// TIA Portal project "灌装完整程序" (V16)

(* hardware
DEVICE "S7-1200 station_1"  S7-1200 Station
   slot 0: "Rack_0"  S7-1200 Rack  Rack  V1.0
   slot 1: "PLC_1"  CPU 1214C DC/DC/DC  6ES7 214-1AG40-0XB0  V4.4
DEVICE "HMI_1"  TP700 Comfort
   slot 0: "HMI_1"  TP700 Comfort  6AV2 124-0GC01-0AX0  16.0.0.0
   slot 1: "HMI_RT_1"  TP700 Comfort  6AV2 124-0GC01-0AX0  16.0.0.0
   slot 5: "HMI_1.IE_CP_1"  PROFINET Interface  16.0.0.0
      slot 1: "PROFINET Interface_1"  PROFINET Interface
         slot 1: "Port_1"  Port
         slot 2: "Port_2"  Port
   slot 7: "HMI_1.MPI/DP_CP_1"  MPI/DP Interface  16.0.0.0
*)

// ===== PLC "PLC_1"  CPU 1214C DC/DC/DC =====

VAR_GLOBAL   // PLC tag table "默认变量表"
   "System_Byte" AT %MB1 : Byte;
   "FirstScan" AT %M1.0 : Bool;
   "DiagStatusUpdate" AT %M1.1 : Bool;
   "AlwaysTRUE" AT %M1.2 : Bool;
   "AlwaysFALSE" AT %M1.3 : Bool;
   "Clock_Byte" AT %MB0 : Byte;
   "Clock_10Hz" AT %M0.0 : Bool;
   "Clock_5Hz" AT %M0.1 : Bool;
   "Clock_2.5Hz" AT %M0.2 : Bool;
   "Clock_2Hz" AT %M0.3 : Bool;
   "Clock_1.25Hz" AT %M0.4 : Bool;
   "Clock_1Hz" AT %M0.5 : Bool;
   "Clock_0.625Hz" AT %M0.6 : Bool;
   "Clock_0.5Hz" AT %M0.7 : Bool;
END_VAR

VAR_GLOBAL   // PLC tag table "I"
   "启动" AT %I0.0 : Bool;
   "停止" AT %I0.1 : Bool;
   "到达称重吹气位置" AT %I0.2 : Bool;
   "到达灌装位置" AT %I0.3 : Bool;
   "到达拧盖位置" AT %I0.4 : Bool;
   "到达包装热缩位置" AT %I0.5 : Bool;
   "到达清洗位置" AT %I0.6 : Bool;
   "到达消毒位置" AT %I0.7 : Bool;
   "到达标签投放位置" AT %I1.0 : Bool;
   "称重检测" AT %IW30 : Int;
   "液位检测" AT %IW32 : Int;
   "吹气气缸上限位" AT %I1.1 : Bool;
   "吹气气缸下限位" AT %I1.2 : Bool;
   "灌装气缸上限位" AT %I1.3 : Bool;
   "灌装气缸下限位" AT %I1.4 : Bool;
   "拧盖气缸上限位" AT %I1.5 : Bool;
   "拧盖气缸下限位" AT %I2.0 : Bool;
   "复位" AT %I2.1 : Bool;
END_VAR

VAR_GLOBAL   // PLC tag table "O"
   "运行指示灯" AT %Q0.0 : Bool;
   "吹气阀门" AT %Q0.1 : Bool;
   "灌装阀门" AT %Q0.2 : Bool;
   "拧盖气缸" AT %Q0.3 : Bool;
   "拧盖电机" AT %Q0.4 : Bool;
   "标签投放" AT %Q0.5 : Bool;
   "包装热缩" AT %Q0.6 : Bool;
   "清洗机" AT %Q0.7 : Bool;
   "消毒机" AT %Q1.0 : Bool;
   "传送带" AT %Q1.1 : Bool;
   "吹气气缸" AT %Q2.0 : Bool;
   "灌装气缸" AT %Q2.1 : Bool;
   "瓶子异常示灯" AT %Q2.2 : Bool;
   "有杂物指示灯" AT %Q2.3 : Bool;
END_VAR

DATA_BLOCK "DB"   // DB1
{ S7_Optimized_Access := 'TRUE' }
VERSION : 0.1
   VAR
      "P/N" : Array[0..100] of Bool;
      仿真数据 : Struct
         仿真开关 : Bool;
         传送带 : Int;
         罐子 : Struct
            X : Int;
            Y : Int;
         END_STRUCT;
         吹气 : Struct
            气缸 : Int;
         END_STRUCT;
         灌装 : Struct
            气缸 : Int;
            液位 : Int;
         END_STRUCT;
         拧盖 : Struct
            盖子显示 : Bool;
            气缸 : Int;
            拧盖进度 : Int;
         END_STRUCT;
         标签投放 : Struct
            大标显示 : Bool;
            小标显示 : Bool;
            标签X : Int;
            标签Y : Int;
            标签Y辅助 : Int;
         END_STRUCT;
         热缩 : Struct
            热缩进度 : Int;
         END_STRUCT;
         清洗 : Struct
            清洗进度 : Int;
         END_STRUCT;
         消毒 : Struct
            消毒进度 : Int;
         END_STRUCT;
      END_STRUCT;
      HMI按键 : Struct
         启动 : Bool;
         停止 : Bool;
         复位 : Bool;
         仿真瓶子质量过低 : Bool;
         仿真瓶子质量超重 : Bool;
      END_STRUCT;
      设定数据 : Struct
         称重质量上限 : Real := 160.0;
         称重质量下限 : Real := 140.0;
         灌装液位 : Int := 85;
      END_STRUCT;
      检测数据 : Struct
         转换值 : Array[0..1] of Real;
         中间值 : Array[0..1] of Real;
         液位实际值 : Real;
         称重实际值 : Real;
         液位仿真值 : Real;
         称重仿真值 : Real;
      END_STRUCT;
      状态 : Struct
         完成吹气 : Bool;
         吹气气缸缩回 : Bool;
         完成灌装 : Bool;
         灌装气缸缩回 : Bool;
         完成拧盖 : Bool;
         拧盖气缸缩回 : Bool;
         标签投放完毕 : Bool;
         热缩完毕 : Bool;
         清洗完毕 : Bool;
         消毒完毕 : Bool;
         流程 : Int;
      END_STRUCT;
   END_VAR
BEGIN
END_DATA_BLOCK

// folder: System blocks/Program resources

DATA_BLOCK "IEC_Timer_0_DB"   // DB2
{ S7_Optimized_Access := 'TRUE' }
AUTHOR : Simatic
FAMILY : IEC
NAME : IEC_TMR
VERSION : 1.0
// stored: InstanceOfName IEC_TIMER
"IEC_TIMER"
BEGIN
END_DATA_BLOCK

DATA_BLOCK "IEC_Timer_0_DB_1"   // DB3
{ S7_Optimized_Access := 'TRUE' }
AUTHOR : Simatic
FAMILY : IEC
NAME : IEC_TMR
VERSION : 1.0
// stored: InstanceOfName IEC_TIMER
"IEC_TIMER"
BEGIN
END_DATA_BLOCK

DATA_BLOCK "IEC_Timer_0_DB_2"   // DB4
{ S7_Optimized_Access := 'TRUE' }
AUTHOR : Simatic
FAMILY : IEC
NAME : IEC_TMR
VERSION : 1.0
// stored: InstanceOfName IEC_TIMER
"IEC_TIMER"
BEGIN
END_DATA_BLOCK

DATA_BLOCK "IEC_Timer_0_DB_3"   // DB5
{ S7_Optimized_Access := 'TRUE' }
AUTHOR : Simatic
FAMILY : IEC
NAME : IEC_TMR
VERSION : 1.0
// stored: InstanceOfName IEC_TIMER
"IEC_TIMER"
BEGIN
END_DATA_BLOCK

DATA_BLOCK "吹气延时"   // DB6
{ S7_Optimized_Access := 'TRUE' }
AUTHOR : Simatic
FAMILY : IEC
NAME : IEC_TMR
VERSION : 1.0
// stored: InstanceOfName IEC_TIMER
"IEC_TIMER"
BEGIN
END_DATA_BLOCK

// folder: (top level)

FUNCTION "04流程" : Void   // FC1, LAD
{ S7_Optimized_Access := 'TRUE' }
VERSION : 0.1
BEGIN

REGION Network 1
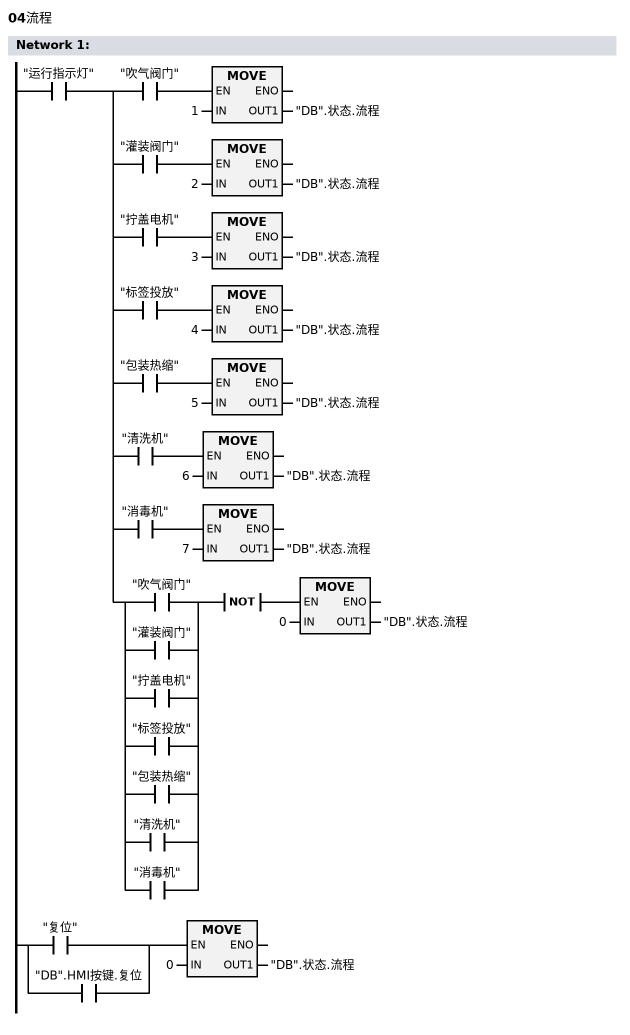
   RUNG wire#powerrail
      Contact( "运行指示灯" )
      wire#w1
      Contact( "吹气阀门" )
      Move(in := 1, out1 => "DB".状态.流程)
   END_RUNG
   RUNG wire#w1
      Contact( "灌装阀门" )
      Move(in := 2, out1 => "DB".状态.流程)
   END_RUNG
   RUNG wire#w1
      Contact( "拧盖电机" )
      Move(in := 3, out1 => "DB".状态.流程)
   END_RUNG
   RUNG wire#w1
      Contact( "标签投放" )
      Move(in := 4, out1 => "DB".状态.流程)
   END_RUNG
   RUNG wire#w1
      Contact( "包装热缩" )
      Move(in := 5, out1 => "DB".状态.流程)
   END_RUNG
   RUNG wire#w1
      Contact( "清洗机" )
      Move(in := 6, out1 => "DB".状态.流程)
   END_RUNG
   RUNG wire#w1
      Contact( "消毒机" )
      Move(in := 7, out1 => "DB".状态.流程)
   END_RUNG
   RUNG wire#w1
      Contact( "吹气阀门" )
      wire#w2
      Not()
      Move(in := 0, out1 => "DB".状态.流程)
   END_RUNG
   RUNG wire#w1
      Contact( "灌装阀门" )
   END_RUNG wire#w2
   RUNG wire#w1
      Contact( "拧盖电机" )
   END_RUNG wire#w2
   RUNG wire#w1
      Contact( "标签投放" )
   END_RUNG wire#w2
   RUNG wire#w1
      Contact( "包装热缩" )
   END_RUNG wire#w2
   RUNG wire#w1
      Contact( "清洗机" )
   END_RUNG wire#w2
   RUNG wire#w1
      Contact( "消毒机" )
   END_RUNG wire#w2
   RUNG wire#powerrail
      Contact( "复位" )
      wire#w3
      Move(in := 0, out1 => "DB".状态.流程)
   END_RUNG
   RUNG wire#powerrail
      Contact( "DB".HMI按键.复位 )
   END_RUNG wire#w3
   // the same network as SCL:
   IF "运行指示灯" AND "吹气阀门" THEN "DB".状态.流程 := 1; END_IF;
   IF "运行指示灯" AND "灌装阀门" THEN "DB".状态.流程 := 2; END_IF;
   IF "运行指示灯" AND "拧盖电机" THEN "DB".状态.流程 := 3; END_IF;
   IF "运行指示灯" AND "标签投放" THEN "DB".状态.流程 := 4; END_IF;
   IF "运行指示灯" AND "包装热缩" THEN "DB".状态.流程 := 5; END_IF;
   IF "运行指示灯" AND "清洗机" THEN "DB".状态.流程 := 6; END_IF;
   IF "运行指示灯" AND "消毒机" THEN "DB".状态.流程 := 7; END_IF;
   IF NOT ("运行指示灯" AND ("吹气阀门" OR "灌装阀门" OR "拧盖电机" OR "标签投放" OR "包装热缩" OR "清洗机" OR "消毒机")) THEN
       "DB".状态.流程 := 0;
   END_IF;
   IF "复位" OR "DB".HMI按键.复位 THEN "DB".状态.流程 := 0; END_IF;
END_REGION
END_FUNCTION

FUNCTION "01系统启停" : Void   // FC2, LAD
{ S7_Optimized_Access := 'TRUE' }
VERSION : 0.1
BEGIN

REGION Network 1
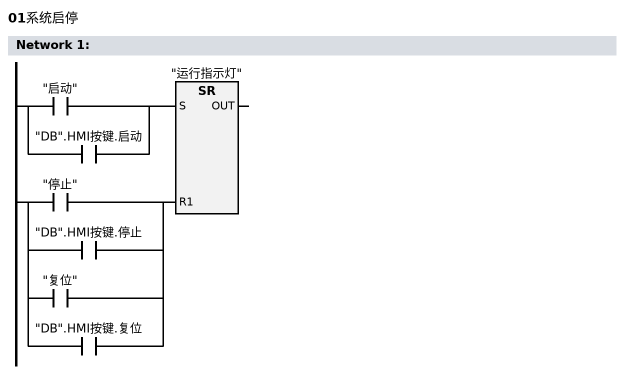
   RUNG wire#powerrail
      Contact( "启动" )
      wire#w1
      S_SR(operand := "运行指示灯", r1 := wire#w2)
   END_RUNG
   RUNG wire#powerrail
      Contact( "DB".HMI按键.启动 )
   END_RUNG wire#w1
   RUNG wire#powerrail
      Contact( "停止" )
   END_RUNG wire#w2
   RUNG wire#powerrail
      Contact( "DB".HMI按键.停止 )
   END_RUNG wire#w2
   RUNG wire#powerrail
      Contact( "复位" )
   END_RUNG wire#w2
   RUNG wire#powerrail
      Contact( "DB".HMI按键.复位 )
   END_RUNG wire#w2
   // the same network as SCL:
   IF "启动" OR "DB".HMI按键.启动 THEN
       "运行指示灯" := TRUE;   // SR flip-flop
   END_IF;
   IF "停止" OR "DB".HMI按键.停止 OR "复位" OR "DB".HMI按键.复位 THEN "运行指示灯" := FALSE; END_IF;
END_REGION
END_FUNCTION

FUNCTION "03自动控制部分" : Void   // FC3, LAD
{ S7_Optimized_Access := 'TRUE' }
VERSION : 0.1
   VAR_TEMP   // added for the SCL form of the ladder/FBD networks
      _w1 : Bool;
      _w2 : Bool;
      _w3 : Bool;
   END_VAR
BEGIN

REGION Network 1
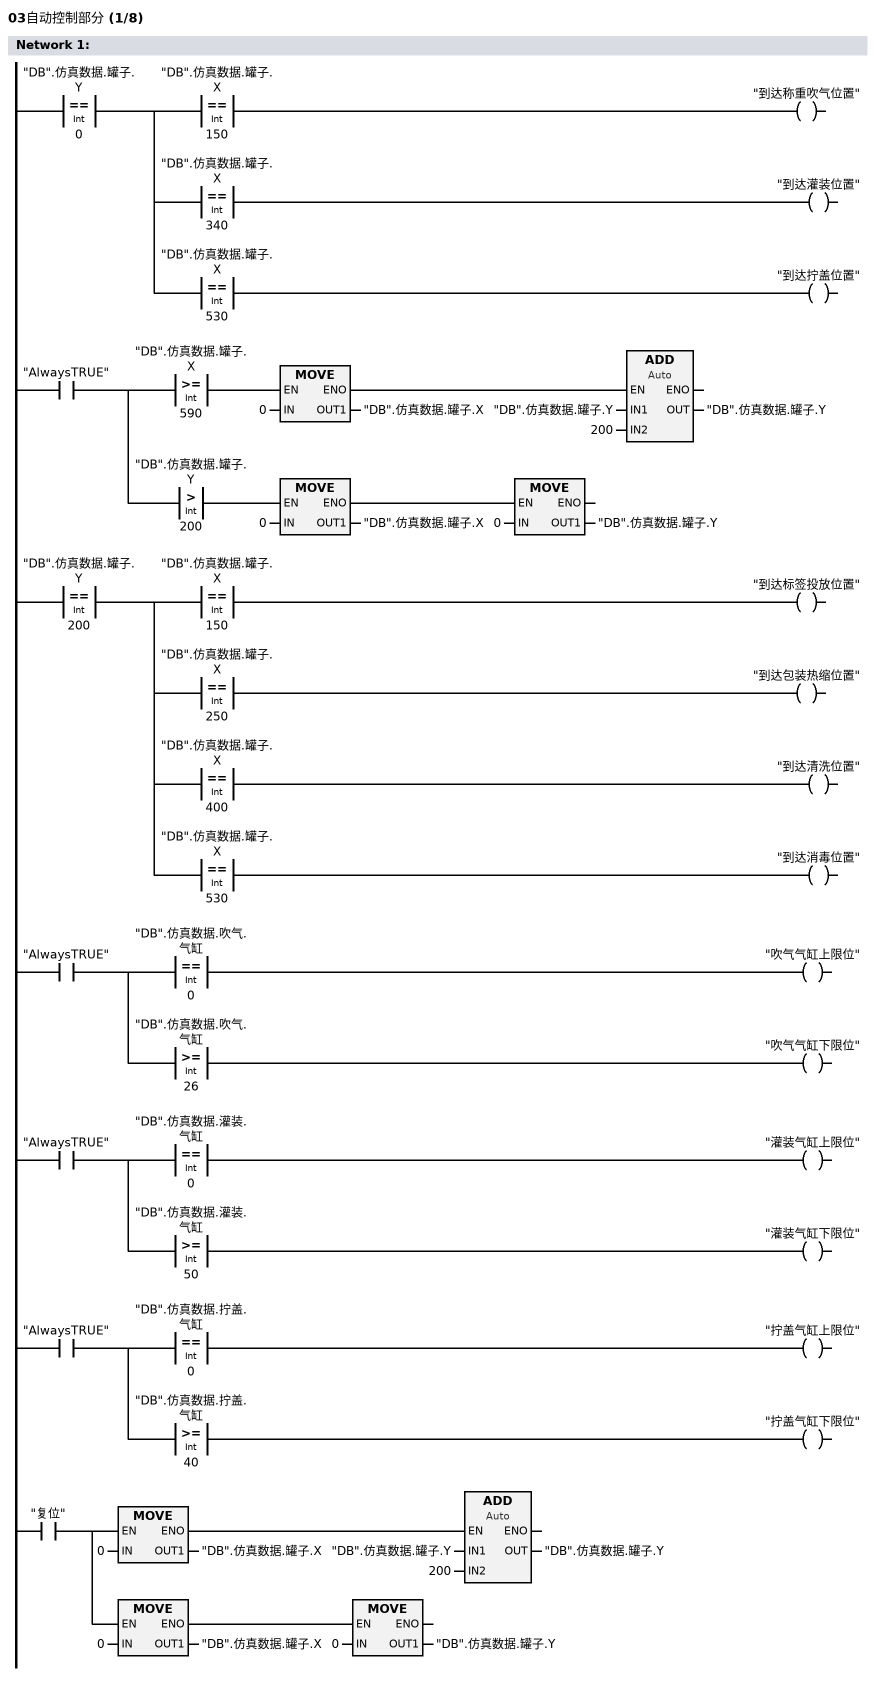
   RUNG wire#powerrail
      { S7_Templates := "SrcType := Int" } EQ_Contact(in1 := "DB".仿真数据.罐子.Y, in2 := 0)
      wire#w1
      { S7_Templates := "SrcType := Int" } EQ_Contact(in1 := "DB".仿真数据.罐子.X, in2 := 150)
      Coil( "到达称重吹气位置" )
   END_RUNG
   RUNG wire#w1
      { S7_Templates := "SrcType := Int" } EQ_Contact(in1 := "DB".仿真数据.罐子.X, in2 := 340)
      Coil( "到达灌装位置" )
   END_RUNG
   RUNG wire#w1
      { S7_Templates := "SrcType := Int" } EQ_Contact(in1 := "DB".仿真数据.罐子.X, in2 := 530)
      Coil( "到达拧盖位置" )
   END_RUNG
   RUNG wire#powerrail
      Contact( "AlwaysTRUE" )
      wire#w2
      { S7_Templates := "SrcType := Int" } GE_Contact(in1 := "DB".仿真数据.罐子.X, in2 := 590)
      Move(in := 0, out1 => "DB".仿真数据.罐子.X)
      Add(in1 := "DB".仿真数据.罐子.Y, in2 := 200, out => "DB".仿真数据.罐子.Y)
   END_RUNG
   RUNG wire#w2
      { S7_Templates := "SrcType := Int" } GT_Contact(in1 := "DB".仿真数据.罐子.Y, in2 := 200)
      Move(in := 0, out1 => "DB".仿真数据.罐子.X)
      Move(in := 0, out1 => "DB".仿真数据.罐子.Y)
   END_RUNG
   RUNG wire#powerrail
      { S7_Templates := "SrcType := Int" } EQ_Contact(in1 := "DB".仿真数据.罐子.Y, in2 := 200)
      wire#w3
      { S7_Templates := "SrcType := Int" } EQ_Contact(in1 := "DB".仿真数据.罐子.X, in2 := 150)
      Coil( "到达标签投放位置" )
   END_RUNG
   RUNG wire#w3
      { S7_Templates := "SrcType := Int" } EQ_Contact(in1 := "DB".仿真数据.罐子.X, in2 := 250)
      Coil( "到达包装热缩位置" )
   END_RUNG
   RUNG wire#w3
      { S7_Templates := "SrcType := Int" } EQ_Contact(in1 := "DB".仿真数据.罐子.X, in2 := 400)
      Coil( "到达清洗位置" )
   END_RUNG
   RUNG wire#w3
      { S7_Templates := "SrcType := Int" } EQ_Contact(in1 := "DB".仿真数据.罐子.X, in2 := 530)
      Coil( "到达消毒位置" )
   END_RUNG
   RUNG wire#powerrail
      Contact( "AlwaysTRUE" )
      wire#w4
      { S7_Templates := "SrcType := Int" } EQ_Contact(in1 := "DB".仿真数据.吹气.气缸, in2 := 0)
      Coil( "吹气气缸上限位" )
   END_RUNG
   RUNG wire#w4
      { S7_Templates := "SrcType := Int" } GE_Contact(in1 := "DB".仿真数据.吹气.气缸, in2 := 26)
      Coil( "吹气气缸下限位" )
   END_RUNG
   RUNG wire#powerrail
      Contact( "AlwaysTRUE" )
      wire#w5
      { S7_Templates := "SrcType := Int" } EQ_Contact(in1 := "DB".仿真数据.灌装.气缸, in2 := 0)
      Coil( "灌装气缸上限位" )
   END_RUNG
   RUNG wire#w5
      { S7_Templates := "SrcType := Int" } GE_Contact(in1 := "DB".仿真数据.灌装.气缸, in2 := 50)
      Coil( "灌装气缸下限位" )
   END_RUNG
   RUNG wire#powerrail
      Contact( "AlwaysTRUE" )
      wire#w6
      { S7_Templates := "SrcType := Int" } EQ_Contact(in1 := "DB".仿真数据.拧盖.气缸, in2 := 0)
      Coil( "拧盖气缸上限位" )
   END_RUNG
   RUNG wire#w6
      { S7_Templates := "SrcType := Int" } GE_Contact(in1 := "DB".仿真数据.拧盖.气缸, in2 := 40)
      Coil( "拧盖气缸下限位" )
   END_RUNG
   RUNG wire#powerrail
      Contact( "复位" )
      wire#w7
      Move(in := 0, out1 => "DB".仿真数据.罐子.X)
      Add(in1 := "DB".仿真数据.罐子.Y, in2 := 200, out => "DB".仿真数据.罐子.Y)
   END_RUNG
   RUNG wire#w7
      Move(in := 0, out1 => "DB".仿真数据.罐子.X)
      Move(in := 0, out1 => "DB".仿真数据.罐子.Y)
   END_RUNG
   // the same network as SCL:
   #_w1 := "DB".仿真数据.罐子.Y = 0;
   "到达称重吹气位置" := #_w1 AND ("DB".仿真数据.罐子.X = 150);
   "到达灌装位置" := #_w1 AND ("DB".仿真数据.罐子.X = 340);
   "到达拧盖位置" := #_w1 AND ("DB".仿真数据.罐子.X = 530);
   #_w2 := "AlwaysTRUE" AND ("DB".仿真数据.罐子.X >= 590);
   IF #_w2 THEN
       "DB".仿真数据.罐子.X := 0;
       "DB".仿真数据.罐子.Y := "DB".仿真数据.罐子.Y + 200;
   END_IF;
   IF "AlwaysTRUE" AND ("DB".仿真数据.罐子.Y > 200) THEN
       "DB".仿真数据.罐子.X := 0;
       "DB".仿真数据.罐子.Y := 0;
   END_IF;
   #_w3 := "DB".仿真数据.罐子.Y = 200;
   "到达标签投放位置" := #_w3 AND ("DB".仿真数据.罐子.X = 150);
   "到达包装热缩位置" := #_w3 AND ("DB".仿真数据.罐子.X = 250);
   "到达清洗位置" := #_w3 AND ("DB".仿真数据.罐子.X = 400);
   "到达消毒位置" := #_w3 AND ("DB".仿真数据.罐子.X = 530);
   "吹气气缸上限位" := "AlwaysTRUE" AND ("DB".仿真数据.吹气.气缸 = 0);
   "吹气气缸下限位" := "AlwaysTRUE" AND ("DB".仿真数据.吹气.气缸 >= 26);
   "灌装气缸上限位" := "AlwaysTRUE" AND ("DB".仿真数据.灌装.气缸 = 0);
   "灌装气缸下限位" := "AlwaysTRUE" AND ("DB".仿真数据.灌装.气缸 >= 50);
   "拧盖气缸上限位" := "AlwaysTRUE" AND ("DB".仿真数据.拧盖.气缸 = 0);
   "拧盖气缸下限位" := "AlwaysTRUE" AND ("DB".仿真数据.拧盖.气缸 >= 40);
   IF "复位" THEN
       "DB".仿真数据.罐子.X := 0;
       "DB".仿真数据.罐子.Y := "DB".仿真数据.罐子.Y + 200;
       "DB".仿真数据.罐子.X := 0;
       "DB".仿真数据.罐子.Y := 0;
   END_IF;
END_REGION

REGION Network 2: 传送带控制
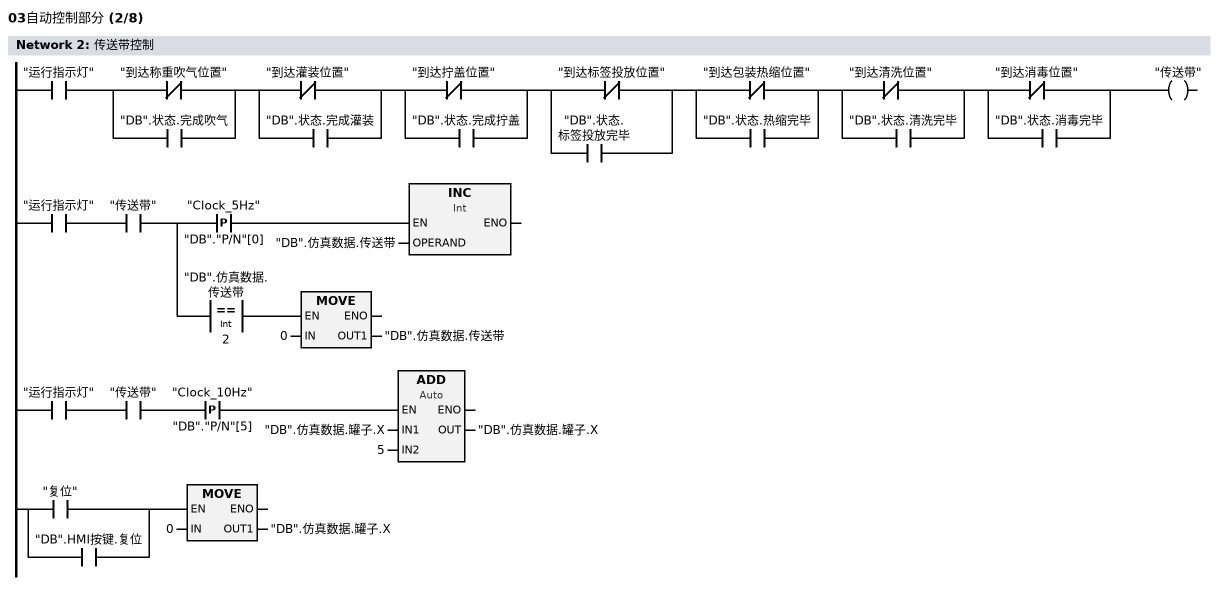
   RUNG wire#powerrail
      Contact( "运行指示灯" )
      wire#w1
      I_Contact( "到达称重吹气位置" )
      wire#w2
      I_Contact( "到达灌装位置" )
      wire#w3
      I_Contact( "到达拧盖位置" )
      wire#w4
      I_Contact( "到达标签投放位置" )
      wire#w5
      I_Contact( "到达包装热缩位置" )
      wire#w6
      I_Contact( "到达清洗位置" )
      wire#w7
      I_Contact( "到达消毒位置" )
      wire#w8
      Coil( "传送带" )
   END_RUNG
   RUNG wire#w1
      Contact( "DB".状态.完成吹气 )
   END_RUNG wire#w2
   RUNG wire#w2
      Contact( "DB".状态.完成灌装 )
   END_RUNG wire#w3
   RUNG wire#w3
      Contact( "DB".状态.完成拧盖 )
   END_RUNG wire#w4
   RUNG wire#w4
      Contact( "DB".状态.标签投放完毕 )
   END_RUNG wire#w5
   RUNG wire#w5
      Contact( "DB".状态.热缩完毕 )
   END_RUNG wire#w6
   RUNG wire#w6
      Contact( "DB".状态.清洗完毕 )
   END_RUNG wire#w7
   RUNG wire#w7
      Contact( "DB".状态.消毒完毕 )
   END_RUNG wire#w8
   RUNG wire#powerrail
      Contact( "运行指示灯" )
      Contact( "传送带" )
      wire#w9
      P_Contact(operand := "Clock_5Hz", bit := "DB"."P/N"[0])
      { S7_Templates := "DestType := Int" } Inc( "DB".仿真数据.传送带 )
   END_RUNG
   RUNG wire#w9
      { S7_Templates := "SrcType := Int" } EQ_Contact(in1 := "DB".仿真数据.传送带, in2 := 2)
      Move(in := 0, out1 => "DB".仿真数据.传送带)
   END_RUNG
   RUNG wire#powerrail
      Contact( "运行指示灯" )
      Contact( "传送带" )
      P_Contact(operand := "Clock_10Hz", bit := "DB"."P/N"[5])
      Add(in1 := "DB".仿真数据.罐子.X, in2 := 5, out => "DB".仿真数据.罐子.X)
   END_RUNG
   RUNG wire#powerrail
      Contact( "复位" )
      wire#w10
      Move(in := 0, out1 => "DB".仿真数据.罐子.X)
   END_RUNG
   RUNG wire#powerrail
      Contact( "DB".HMI按键.复位 )
   END_RUNG wire#w10
   // the same network as SCL:
   "传送带" := "运行指示灯" AND (NOT "到达称重吹气位置" OR "DB".状态.完成吹气) AND (NOT "到达灌装位置" OR "DB".状态.完成灌装) AND (NOT "到达拧盖位置" OR "DB".状态.完成拧盖) AND (NOT "到达标签投放位置" OR "DB".状态.标签投放完毕) AND (NOT "到达包装热缩位置" OR "DB".状态.热缩完毕) AND (NOT "到达清洗位置" OR "DB".状态.清洗完毕) AND (NOT "到达消毒位置" OR "DB".状态.消毒完毕);
   #_w1 := "运行指示灯" AND "传送带";
   #_w2 := #_w1 AND "Clock_5Hz" AND NOT "DB"."P/N"[0];   // rising edge of "Clock_5Hz"
   "DB"."P/N"[0] := "Clock_5Hz";
   IF #_w2 THEN "DB".仿真数据.传送带 := "DB".仿真数据.传送带 + 1; END_IF;
   IF #_w1 AND ("DB".仿真数据.传送带 = 2) THEN "DB".仿真数据.传送带 := 0; END_IF;
   #_w3 := "运行指示灯" AND "传送带" AND "Clock_10Hz" AND NOT "DB"."P/N"[5];   // rising edge of "Clock_10Hz"
   "DB"."P/N"[5] := "Clock_10Hz";
   IF #_w3 THEN "DB".仿真数据.罐子.X := "DB".仿真数据.罐子.X + 5; END_IF;
   IF "复位" OR "DB".HMI按键.复位 THEN "DB".仿真数据.罐子.X := 0; END_IF;
END_REGION

REGION Network 3: 称重吹气
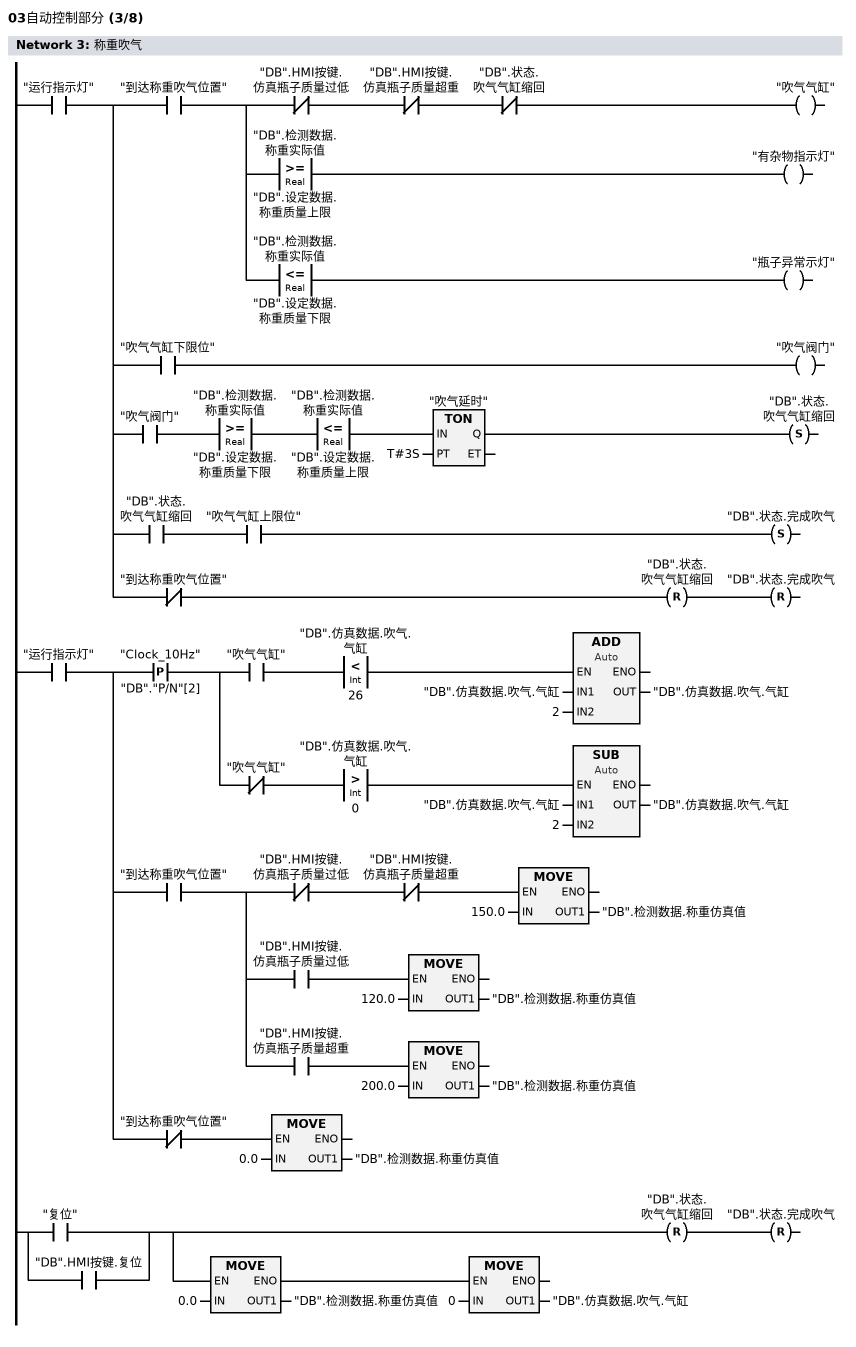
   #_w1 := "运行指示灯" AND "到达称重吹气位置";
   "吹气气缸" := #_w1 AND NOT "DB".HMI按键.仿真瓶子质量过低 AND NOT "DB".HMI按键.仿真瓶子质量超重 AND NOT "DB".状态.吹气气缸缩回;
   "有杂物指示灯" := #_w1 AND ("DB".检测数据.称重实际值 >= "DB".设定数据.称重质量上限);
   "瓶子异常示灯" := #_w1 AND ("DB".检测数据.称重实际值 <= "DB".设定数据.称重质量下限);
   "吹气阀门" := "运行指示灯" AND "吹气气缸下限位";
   "吹气延时".TON(IN := "运行指示灯" AND "吹气阀门" AND ("DB".检测数据.称重实际值 >= "DB".设定数据.称重质量下限) AND ("DB".检测数据.称重实际值 <= "DB".设定数据.称重质量上限),
              PT := T#3S);
   IF "吹气延时".Q THEN "DB".状态.吹气气缸缩回 := TRUE; END_IF;
   IF "运行指示灯" AND "DB".状态.吹气气缸缩回 AND "吹气气缸上限位" THEN "DB".状态.完成吹气 := TRUE; END_IF;
   IF "运行指示灯" AND NOT "到达称重吹气位置" THEN
       "DB".状态.吹气气缸缩回 := FALSE;
       "DB".状态.完成吹气 := FALSE;
   END_IF;
   #_w2 := "运行指示灯" AND "Clock_10Hz" AND NOT "DB"."P/N"[2];   // rising edge of "Clock_10Hz"
   "DB"."P/N"[2] := "Clock_10Hz";
   IF #_w2 AND "吹气气缸" AND ("DB".仿真数据.吹气.气缸 < 26) THEN "DB".仿真数据.吹气.气缸 := "DB".仿真数据.吹气.气缸 + 2; END_IF;
   IF #_w2 AND NOT "吹气气缸" AND ("DB".仿真数据.吹气.气缸 > 0) THEN "DB".仿真数据.吹气.气缸 := "DB".仿真数据.吹气.气缸 - 2; END_IF;
   #_w3 := "运行指示灯" AND "到达称重吹气位置";
   IF #_w3 AND NOT "DB".HMI按键.仿真瓶子质量过低 AND NOT "DB".HMI按键.仿真瓶子质量超重 THEN "DB".检测数据.称重仿真值 := 150.0; END_IF;
   IF #_w3 AND "DB".HMI按键.仿真瓶子质量过低 THEN "DB".检测数据.称重仿真值 := 120.0; END_IF;
   IF #_w3 AND "DB".HMI按键.仿真瓶子质量超重 THEN "DB".检测数据.称重仿真值 := 200.0; END_IF;
   IF "运行指示灯" AND NOT "到达称重吹气位置" THEN "DB".检测数据.称重仿真值 := 0.0; END_IF;
   IF "复位" OR "DB".HMI按键.复位 THEN
       "DB".状态.吹气气缸缩回 := FALSE;
       "DB".状态.完成吹气 := FALSE;
       "DB".检测数据.称重仿真值 := 0.0;
       "DB".仿真数据.吹气.气缸 := 0;
   END_IF;
END_REGION

REGION Network 4: 灌装
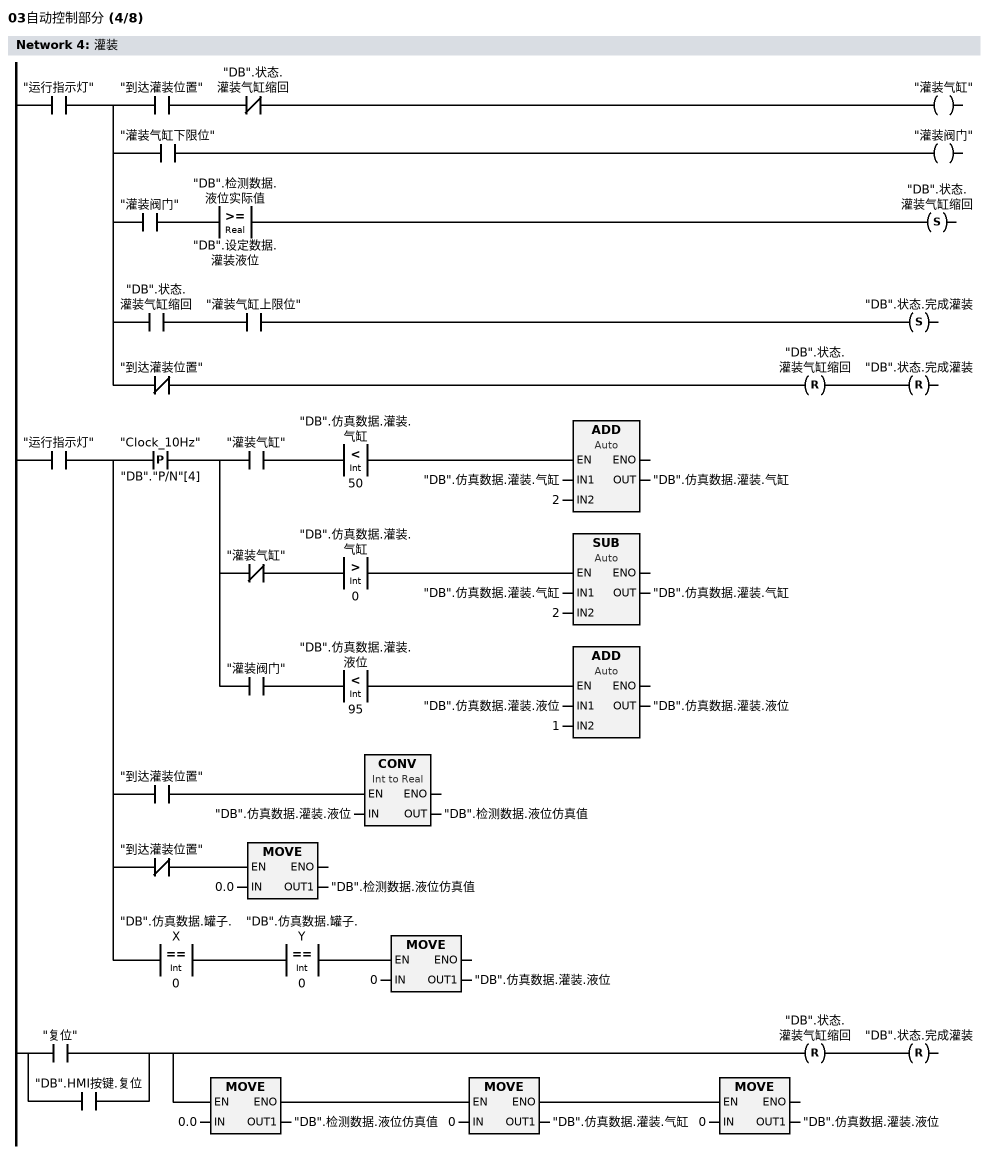
   RUNG wire#powerrail
      Contact( "运行指示灯" )
      wire#w1
      Contact( "到达灌装位置" )
      I_Contact( "DB".状态.灌装气缸缩回 )
      Coil( "灌装气缸" )
   END_RUNG
   RUNG wire#w1
      Contact( "灌装气缸下限位" )
      Coil( "灌装阀门" )
   END_RUNG
   RUNG wire#w1
      Contact( "灌装阀门" )
      { S7_Templates := "SrcType := Real" } GE_Contact(in1 := "DB".检测数据.液位实际值, in2 := "DB".设定数据.灌装液位)
      S_Coil( "DB".状态.灌装气缸缩回 )
   END_RUNG
   RUNG wire#w1
      Contact( "DB".状态.灌装气缸缩回 )
      Contact( "灌装气缸上限位" )
      S_Coil( "DB".状态.完成灌装 )
   END_RUNG
   RUNG wire#w1
      I_Contact( "到达灌装位置" )
      R_Coil( "DB".状态.灌装气缸缩回 )
      R_Coil( "DB".状态.完成灌装 )
   END_RUNG
   RUNG wire#powerrail
      Contact( "运行指示灯" )
      wire#w2
      P_Contact(operand := "Clock_10Hz", bit := "DB"."P/N"[4])
      wire#w3
      Contact( "灌装气缸" )
      { S7_Templates := "SrcType := Int" } LT_Contact(in1 := "DB".仿真数据.灌装.气缸, in2 := 50)
      Add(in1 := "DB".仿真数据.灌装.气缸, in2 := 2, out => "DB".仿真数据.灌装.气缸)
   END_RUNG
   RUNG wire#w3
      I_Contact( "灌装气缸" )
      { S7_Templates := "SrcType := Int" } GT_Contact(in1 := "DB".仿真数据.灌装.气缸, in2 := 0)
      Sub(in1 := "DB".仿真数据.灌装.气缸, in2 := 2, out => "DB".仿真数据.灌装.气缸)
   END_RUNG
   RUNG wire#w3
      Contact( "灌装阀门" )
      { S7_Templates := "SrcType := Int" } LT_Contact(in1 := "DB".仿真数据.灌装.液位, in2 := 95)
      Add(in1 := "DB".仿真数据.灌装.液位, in2 := 1, out => "DB".仿真数据.灌装.液位)
   END_RUNG
   RUNG wire#w2
      Contact( "到达灌装位置" )
      { S7_Templates := "[SrcType := Int, DestType := Real]" } Convert(in := "DB".仿真数据.灌装.液位, out => "DB".检测数据.液位仿真值)
   END_RUNG
   RUNG wire#w2
      I_Contact( "到达灌装位置" )
      Move(in := 0.0, out1 => "DB".检测数据.液位仿真值)
   END_RUNG
   RUNG wire#w2
      { S7_Templates := "SrcType := Int" } EQ_Contact(in1 := "DB".仿真数据.罐子.X, in2 := 0)
      { S7_Templates := "SrcType := Int" } EQ_Contact(in1 := "DB".仿真数据.罐子.Y, in2 := 0)
      Move(in := 0, out1 => "DB".仿真数据.灌装.液位)
   END_RUNG
   RUNG wire#powerrail
      Contact( "复位" )
      wire#w4
      R_Coil( "DB".状态.灌装气缸缩回 )
      R_Coil( "DB".状态.完成灌装 )
   END_RUNG
   RUNG wire#powerrail
      Contact( "DB".HMI按键.复位 )
   END_RUNG wire#w4
   RUNG wire#w4
      Move(in := 0.0, out1 => "DB".检测数据.液位仿真值)
      Move(in := 0, out1 => "DB".仿真数据.灌装.气缸)
      Move(in := 0, out1 => "DB".仿真数据.灌装.液位)
   END_RUNG
   // the same network as SCL:
   "灌装气缸" := "运行指示灯" AND "到达灌装位置" AND NOT "DB".状态.灌装气缸缩回;
   "灌装阀门" := "运行指示灯" AND "灌装气缸下限位";
   IF "运行指示灯" AND "灌装阀门" AND ("DB".检测数据.液位实际值 >= "DB".设定数据.灌装液位) THEN "DB".状态.灌装气缸缩回 := TRUE; END_IF;
   IF "运行指示灯" AND "DB".状态.灌装气缸缩回 AND "灌装气缸上限位" THEN "DB".状态.完成灌装 := TRUE; END_IF;
   IF "运行指示灯" AND NOT "到达灌装位置" THEN
       "DB".状态.灌装气缸缩回 := FALSE;
       "DB".状态.完成灌装 := FALSE;
   END_IF;
   #_w1 := "运行指示灯" AND "Clock_10Hz" AND NOT "DB"."P/N"[4];   // rising edge of "Clock_10Hz"
   "DB"."P/N"[4] := "Clock_10Hz";
   IF #_w1 AND "灌装气缸" AND ("DB".仿真数据.灌装.气缸 < 50) THEN "DB".仿真数据.灌装.气缸 := "DB".仿真数据.灌装.气缸 + 2; END_IF;
   IF #_w1 AND NOT "灌装气缸" AND ("DB".仿真数据.灌装.气缸 > 0) THEN "DB".仿真数据.灌装.气缸 := "DB".仿真数据.灌装.气缸 - 2; END_IF;
   IF #_w1 AND "灌装阀门" AND ("DB".仿真数据.灌装.液位 < 95) THEN "DB".仿真数据.灌装.液位 := "DB".仿真数据.灌装.液位 + 1; END_IF;
   IF "运行指示灯" AND "到达灌装位置" THEN "DB".检测数据.液位仿真值 := INT_TO_REAL("DB".仿真数据.灌装.液位); END_IF;
   IF "运行指示灯" AND NOT "到达灌装位置" THEN "DB".检测数据.液位仿真值 := 0.0; END_IF;
   IF "运行指示灯" AND ("DB".仿真数据.罐子.X = 0) AND ("DB".仿真数据.罐子.Y = 0) THEN "DB".仿真数据.灌装.液位 := 0; END_IF;
   IF "复位" OR "DB".HMI按键.复位 THEN
       "DB".状态.灌装气缸缩回 := FALSE;
       "DB".状态.完成灌装 := FALSE;
       "DB".检测数据.液位仿真值 := 0.0;
       "DB".仿真数据.灌装.气缸 := 0;
       "DB".仿真数据.灌装.液位 := 0;
   END_IF;
END_REGION

REGION Network 5: 拧盖
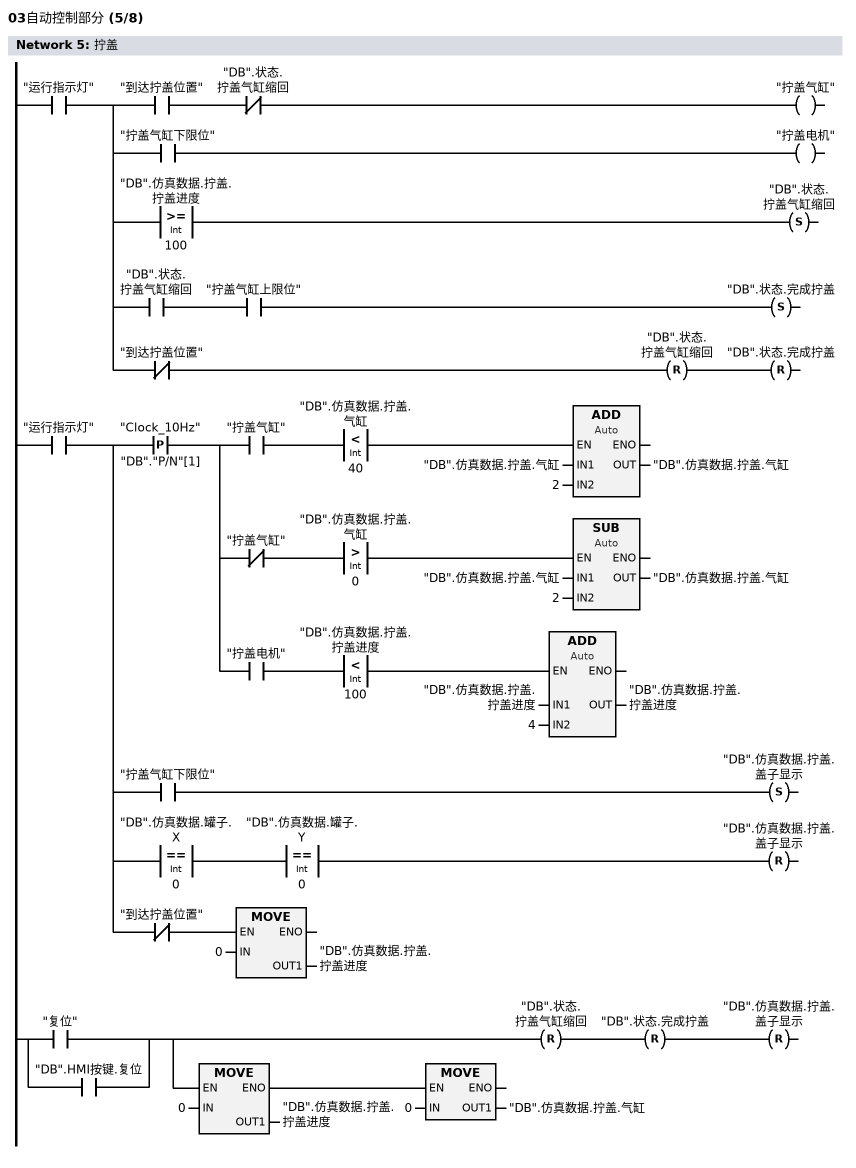
   RUNG wire#powerrail
      Contact( "运行指示灯" )
      wire#w1
      Contact( "到达拧盖位置" )
      I_Contact( "DB".状态.拧盖气缸缩回 )
      Coil( "拧盖气缸" )
   END_RUNG
   RUNG wire#w1
      Contact( "拧盖气缸下限位" )
      Coil( "拧盖电机" )
   END_RUNG
   RUNG wire#w1
      { S7_Templates := "SrcType := Int" } GE_Contact(in1 := "DB".仿真数据.拧盖.拧盖进度, in2 := 100)
      S_Coil( "DB".状态.拧盖气缸缩回 )
   END_RUNG
   RUNG wire#w1
      Contact( "DB".状态.拧盖气缸缩回 )
      Contact( "拧盖气缸上限位" )
      S_Coil( "DB".状态.完成拧盖 )
   END_RUNG
   RUNG wire#w1
      I_Contact( "到达拧盖位置" )
      R_Coil( "DB".状态.拧盖气缸缩回 )
      R_Coil( "DB".状态.完成拧盖 )
   END_RUNG
   RUNG wire#powerrail
      Contact( "运行指示灯" )
      wire#w2
      P_Contact(operand := "Clock_10Hz", bit := "DB"."P/N"[1])
      wire#w3
      Contact( "拧盖气缸" )
      { S7_Templates := "SrcType := Int" } LT_Contact(in1 := "DB".仿真数据.拧盖.气缸, in2 := 40)
      Add(in1 := "DB".仿真数据.拧盖.气缸, in2 := 2, out => "DB".仿真数据.拧盖.气缸)
   END_RUNG
   RUNG wire#w3
      I_Contact( "拧盖气缸" )
      { S7_Templates := "SrcType := Int" } GT_Contact(in1 := "DB".仿真数据.拧盖.气缸, in2 := 0)
      Sub(in1 := "DB".仿真数据.拧盖.气缸, in2 := 2, out => "DB".仿真数据.拧盖.气缸)
   END_RUNG
   RUNG wire#w3
      Contact( "拧盖电机" )
      { S7_Templates := "SrcType := Int" } LT_Contact(in1 := "DB".仿真数据.拧盖.拧盖进度, in2 := 100)
      Add(in1 := "DB".仿真数据.拧盖.拧盖进度, in2 := 4, out => "DB".仿真数据.拧盖.拧盖进度)
   END_RUNG
   RUNG wire#w2
      Contact( "拧盖气缸下限位" )
      S_Coil( "DB".仿真数据.拧盖.盖子显示 )
   END_RUNG
   RUNG wire#w2
      { S7_Templates := "SrcType := Int" } EQ_Contact(in1 := "DB".仿真数据.罐子.X, in2 := 0)
      { S7_Templates := "SrcType := Int" } EQ_Contact(in1 := "DB".仿真数据.罐子.Y, in2 := 0)
      R_Coil( "DB".仿真数据.拧盖.盖子显示 )
   END_RUNG
   RUNG wire#w2
      I_Contact( "到达拧盖位置" )
      Move(in := 0, out1 => "DB".仿真数据.拧盖.拧盖进度)
   END_RUNG
   RUNG wire#powerrail
      Contact( "复位" )
      wire#w4
      R_Coil( "DB".状态.拧盖气缸缩回 )
      R_Coil( "DB".状态.完成拧盖 )
      R_Coil( "DB".仿真数据.拧盖.盖子显示 )
   END_RUNG
   RUNG wire#powerrail
      Contact( "DB".HMI按键.复位 )
   END_RUNG wire#w4
   RUNG wire#w4
      Move(in := 0, out1 => "DB".仿真数据.拧盖.拧盖进度)
      Move(in := 0, out1 => "DB".仿真数据.拧盖.气缸)
   END_RUNG
   // the same network as SCL:
   "拧盖气缸" := "运行指示灯" AND "到达拧盖位置" AND NOT "DB".状态.拧盖气缸缩回;
   "拧盖电机" := "运行指示灯" AND "拧盖气缸下限位";
   IF "运行指示灯" AND ("DB".仿真数据.拧盖.拧盖进度 >= 100) THEN "DB".状态.拧盖气缸缩回 := TRUE; END_IF;
   IF "运行指示灯" AND "DB".状态.拧盖气缸缩回 AND "拧盖气缸上限位" THEN "DB".状态.完成拧盖 := TRUE; END_IF;
   IF "运行指示灯" AND NOT "到达拧盖位置" THEN
       "DB".状态.拧盖气缸缩回 := FALSE;
       "DB".状态.完成拧盖 := FALSE;
   END_IF;
   #_w1 := "运行指示灯" AND "Clock_10Hz" AND NOT "DB"."P/N"[1];   // rising edge of "Clock_10Hz"
   "DB"."P/N"[1] := "Clock_10Hz";
   IF #_w1 AND "拧盖气缸" AND ("DB".仿真数据.拧盖.气缸 < 40) THEN "DB".仿真数据.拧盖.气缸 := "DB".仿真数据.拧盖.气缸 + 2; END_IF;
   IF #_w1 AND NOT "拧盖气缸" AND ("DB".仿真数据.拧盖.气缸 > 0) THEN "DB".仿真数据.拧盖.气缸 := "DB".仿真数据.拧盖.气缸 - 2; END_IF;
   IF #_w1 AND "拧盖电机" AND ("DB".仿真数据.拧盖.拧盖进度 < 100) THEN "DB".仿真数据.拧盖.拧盖进度 := "DB".仿真数据.拧盖.拧盖进度 + 4; END_IF;
   IF "运行指示灯" AND "拧盖气缸下限位" THEN "DB".仿真数据.拧盖.盖子显示 := TRUE; END_IF;
   IF "运行指示灯" AND ("DB".仿真数据.罐子.X = 0) AND ("DB".仿真数据.罐子.Y = 0) THEN "DB".仿真数据.拧盖.盖子显示 := FALSE; END_IF;
   IF "运行指示灯" AND NOT "到达拧盖位置" THEN "DB".仿真数据.拧盖.拧盖进度 := 0; END_IF;
   IF "复位" OR "DB".HMI按键.复位 THEN
       "DB".状态.拧盖气缸缩回 := FALSE;
       "DB".状态.完成拧盖 := FALSE;
       "DB".仿真数据.拧盖.盖子显示 := FALSE;
       "DB".仿真数据.拧盖.拧盖进度 := 0;
       "DB".仿真数据.拧盖.气缸 := 0;
   END_IF;
END_REGION

REGION Network 6: 标签投放
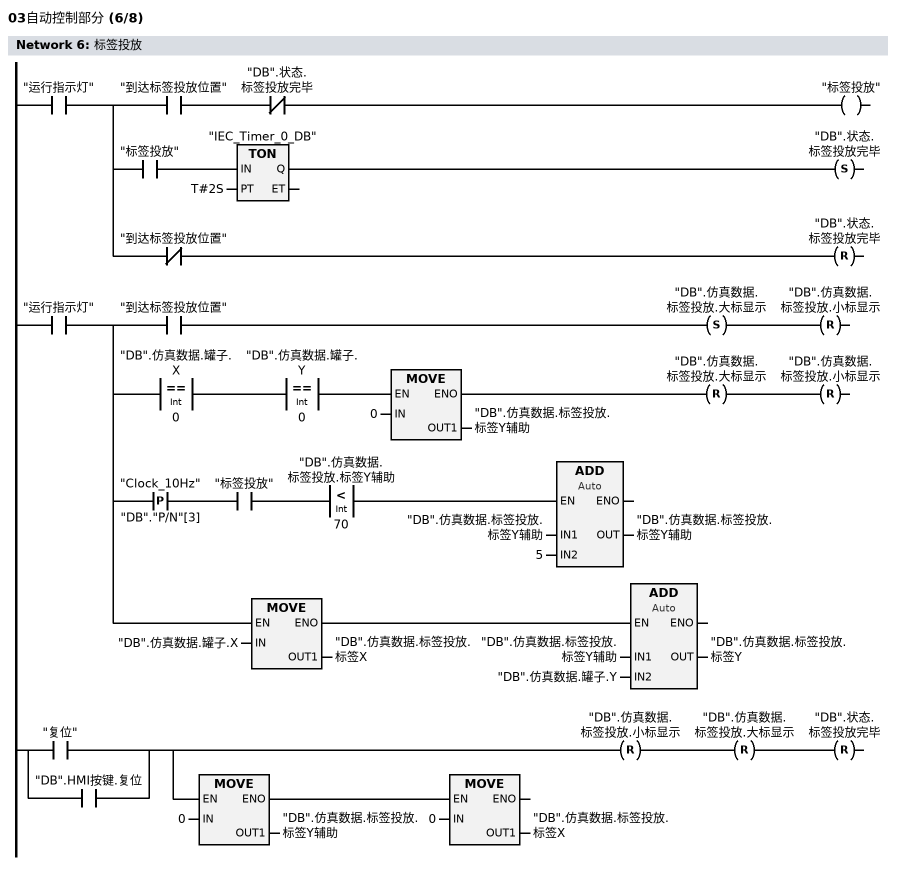
   "标签投放" := "运行指示灯" AND "到达标签投放位置" AND NOT "DB".状态.标签投放完毕;
   "IEC_Timer_0_DB".TON(IN := "运行指示灯" AND "标签投放", PT := T#2S);
   IF "IEC_Timer_0_DB".Q THEN "DB".状态.标签投放完毕 := TRUE; END_IF;
   IF "运行指示灯" AND NOT "到达标签投放位置" THEN "DB".状态.标签投放完毕 := FALSE; END_IF;
   IF "运行指示灯" AND "到达标签投放位置" THEN
       "DB".仿真数据.标签投放.大标显示 := TRUE;
       "DB".仿真数据.标签投放.小标显示 := FALSE;
   END_IF;
   IF "运行指示灯" AND ("DB".仿真数据.罐子.X = 0) AND ("DB".仿真数据.罐子.Y = 0) THEN
       "DB".仿真数据.标签投放.标签Y辅助 := 0;
       "DB".仿真数据.标签投放.大标显示 := FALSE;
       "DB".仿真数据.标签投放.小标显示 := FALSE;
   END_IF;
   #_w1 := "运行指示灯" AND "Clock_10Hz" AND NOT "DB"."P/N"[3];   // rising edge of "Clock_10Hz"
   "DB"."P/N"[3] := "Clock_10Hz";
   IF #_w1 AND "标签投放" AND ("DB".仿真数据.标签投放.标签Y辅助 < 70) THEN
       "DB".仿真数据.标签投放.标签Y辅助 := "DB".仿真数据.标签投放.标签Y辅助 + 5;
   END_IF;
   IF "运行指示灯" THEN
       "DB".仿真数据.标签投放.标签X := "DB".仿真数据.罐子.X;
       "DB".仿真数据.标签投放.标签Y := "DB".仿真数据.标签投放.标签Y辅助 + "DB".仿真数据.罐子.Y;
   END_IF;
   IF "复位" OR "DB".HMI按键.复位 THEN
       "DB".仿真数据.标签投放.小标显示 := FALSE;
       "DB".仿真数据.标签投放.大标显示 := FALSE;
       "DB".状态.标签投放完毕 := FALSE;
       "DB".仿真数据.标签投放.标签Y辅助 := 0;
       "DB".仿真数据.标签投放.标签X := 0;
   END_IF;
END_REGION

REGION Network 7: 包装热缩
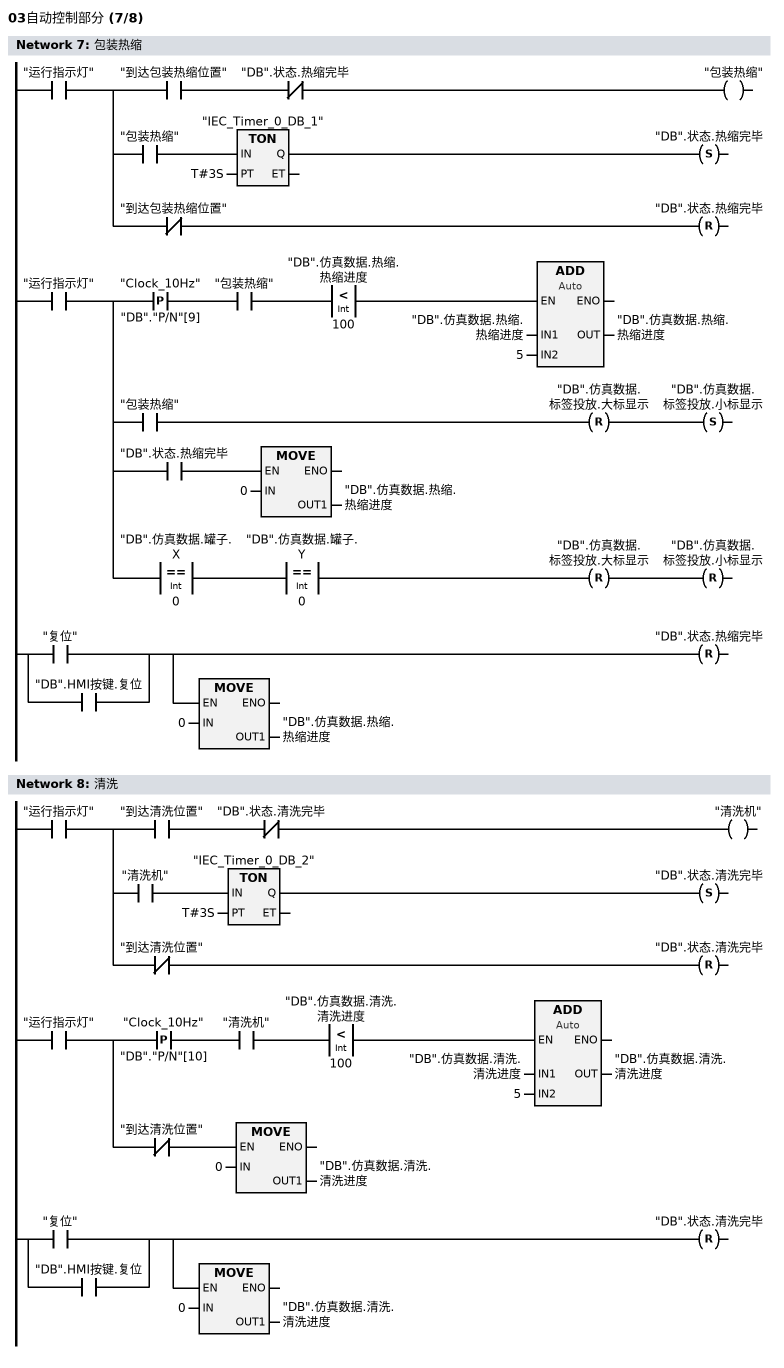
   "包装热缩" := "运行指示灯" AND "到达包装热缩位置" AND NOT "DB".状态.热缩完毕;
   "IEC_Timer_0_DB_1".TON(IN := "运行指示灯" AND "包装热缩", PT := T#3S);
   IF "IEC_Timer_0_DB_1".Q THEN "DB".状态.热缩完毕 := TRUE; END_IF;
   IF "运行指示灯" AND NOT "到达包装热缩位置" THEN "DB".状态.热缩完毕 := FALSE; END_IF;
   #_w1 := "运行指示灯" AND "Clock_10Hz" AND NOT "DB"."P/N"[9];   // rising edge of "Clock_10Hz"
   "DB"."P/N"[9] := "Clock_10Hz";
   IF #_w1 AND "包装热缩" AND ("DB".仿真数据.热缩.热缩进度 < 100) THEN "DB".仿真数据.热缩.热缩进度 := "DB".仿真数据.热缩.热缩进度 + 5; END_IF;
   IF "运行指示灯" AND "包装热缩" THEN
       "DB".仿真数据.标签投放.大标显示 := FALSE;
       "DB".仿真数据.标签投放.小标显示 := TRUE;
   END_IF;
   IF "运行指示灯" AND "DB".状态.热缩完毕 THEN "DB".仿真数据.热缩.热缩进度 := 0; END_IF;
   IF "运行指示灯" AND ("DB".仿真数据.罐子.X = 0) AND ("DB".仿真数据.罐子.Y = 0) THEN
       "DB".仿真数据.标签投放.大标显示 := FALSE;
       "DB".仿真数据.标签投放.小标显示 := FALSE;
   END_IF;
   IF "复位" OR "DB".HMI按键.复位 THEN
       "DB".状态.热缩完毕 := FALSE;
       "DB".仿真数据.热缩.热缩进度 := 0;
   END_IF;
END_REGION

REGION Network 8: 清洗
   "清洗机" := "运行指示灯" AND "到达清洗位置" AND NOT "DB".状态.清洗完毕;
   "IEC_Timer_0_DB_2".TON(IN := "运行指示灯" AND "清洗机", PT := T#3S);
   IF "IEC_Timer_0_DB_2".Q THEN "DB".状态.清洗完毕 := TRUE; END_IF;
   IF "运行指示灯" AND NOT "到达清洗位置" THEN "DB".状态.清洗完毕 := FALSE; END_IF;
   #_w1 := "运行指示灯" AND "Clock_10Hz" AND NOT "DB"."P/N"[10];   // rising edge of "Clock_10Hz"
   "DB"."P/N"[10] := "Clock_10Hz";
   IF #_w1 AND "清洗机" AND ("DB".仿真数据.清洗.清洗进度 < 100) THEN "DB".仿真数据.清洗.清洗进度 := "DB".仿真数据.清洗.清洗进度 + 5; END_IF;
   IF "运行指示灯" AND NOT "到达清洗位置" THEN "DB".仿真数据.清洗.清洗进度 := 0; END_IF;
   IF "复位" OR "DB".HMI按键.复位 THEN
       "DB".状态.清洗完毕 := FALSE;
       "DB".仿真数据.清洗.清洗进度 := 0;
   END_IF;
END_REGION

REGION Network 9: 消毒
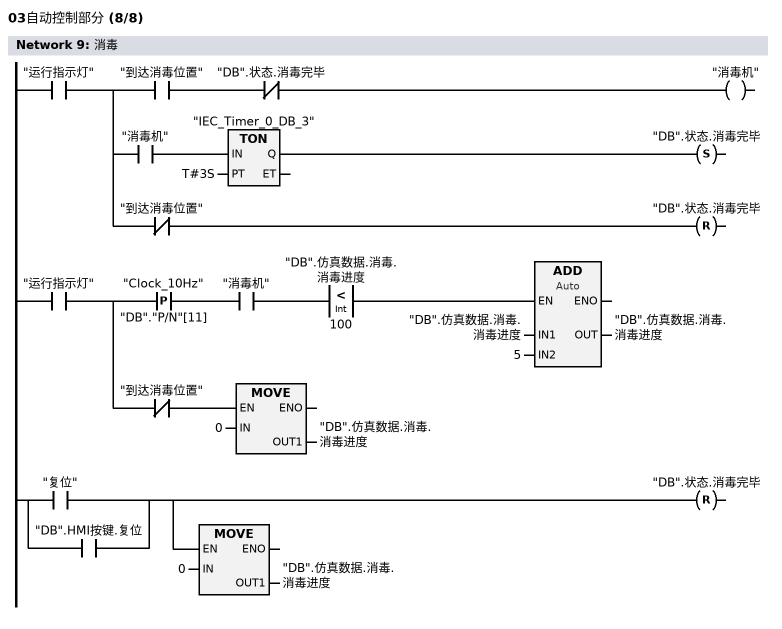
   "消毒机" := "运行指示灯" AND "到达消毒位置" AND NOT "DB".状态.消毒完毕;
   "IEC_Timer_0_DB_3".TON(IN := "运行指示灯" AND "消毒机", PT := T#3S);
   IF "IEC_Timer_0_DB_3".Q THEN "DB".状态.消毒完毕 := TRUE; END_IF;
   IF "运行指示灯" AND NOT "到达消毒位置" THEN "DB".状态.消毒完毕 := FALSE; END_IF;
   #_w1 := "运行指示灯" AND "Clock_10Hz" AND NOT "DB"."P/N"[11];   // rising edge of "Clock_10Hz"
   "DB"."P/N"[11] := "Clock_10Hz";
   IF #_w1 AND "消毒机" AND ("DB".仿真数据.消毒.消毒进度 < 100) THEN "DB".仿真数据.消毒.消毒进度 := "DB".仿真数据.消毒.消毒进度 + 5; END_IF;
   IF "运行指示灯" AND NOT "到达消毒位置" THEN "DB".仿真数据.消毒.消毒进度 := 0; END_IF;
   IF "复位" OR "DB".HMI按键.复位 THEN
       "DB".状态.消毒完毕 := FALSE;
       "DB".仿真数据.消毒.消毒进度 := 0;
   END_IF;
END_REGION
END_FUNCTION

FUNCTION "02模拟量处理" : Void   // FC4, LAD
{ S7_Optimized_Access := 'TRUE' }
VERSION : 0.1
BEGIN

REGION Network 1
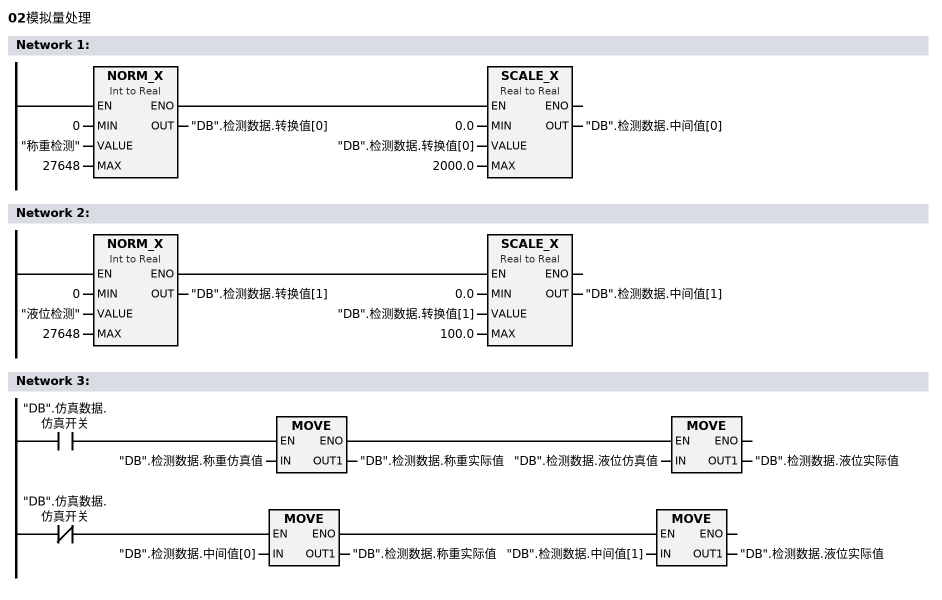
   RUNG wire#powerrail
      { S7_Templates := "[SrcType := Int, DestType := Real]" } Normalize(min := 0, value := "称重检测", max := 27648, out => "DB".检测数据.转换值[0])
      { S7_Templates := "[SrcType := Real, DestType := Real]" } Scale(min := 0.0, value := "DB".检测数据.转换值[0], max := 2000.0, out => "DB".检测数据.中间值[0])
   END_RUNG
   // the same network as SCL:
   "DB".检测数据.转换值[0] := NORM_X(MIN := 0, VALUE := "称重检测", MAX := 27648);
   "DB".检测数据.中间值[0] := SCALE_X(MIN := 0.0, VALUE := "DB".检测数据.转换值[0], MAX := 2000.0);
END_REGION

REGION Network 2
   RUNG wire#powerrail
      { S7_Templates := "[SrcType := Int, DestType := Real]" } Normalize(min := 0, value := "液位检测", max := 27648, out => "DB".检测数据.转换值[1])
      { S7_Templates := "[SrcType := Real, DestType := Real]" } Scale(min := 0.0, value := "DB".检测数据.转换值[1], max := 100.0, out => "DB".检测数据.中间值[1])
   END_RUNG
   // the same network as SCL:
   "DB".检测数据.转换值[1] := NORM_X(MIN := 0, VALUE := "液位检测", MAX := 27648);
   "DB".检测数据.中间值[1] := SCALE_X(MIN := 0.0, VALUE := "DB".检测数据.转换值[1], MAX := 100.0);
END_REGION

REGION Network 3
   RUNG wire#powerrail
      Contact( "DB".仿真数据.仿真开关 )
      Move(in := "DB".检测数据.称重仿真值, out1 => "DB".检测数据.称重实际值)
      Move(in := "DB".检测数据.液位仿真值, out1 => "DB".检测数据.液位实际值)
   END_RUNG
   RUNG wire#powerrail
      I_Contact( "DB".仿真数据.仿真开关 )
      Move(in := "DB".检测数据.中间值[0], out1 => "DB".检测数据.称重实际值)
      Move(in := "DB".检测数据.中间值[1], out1 => "DB".检测数据.液位实际值)
   END_RUNG
   // the same network as SCL:
   IF "DB".仿真数据.仿真开关 THEN
       "DB".检测数据.称重实际值 := "DB".检测数据.称重仿真值;
       "DB".检测数据.液位实际值 := "DB".检测数据.液位仿真值;
   END_IF;
   IF NOT "DB".仿真数据.仿真开关 THEN
       "DB".检测数据.称重实际值 := "DB".检测数据.中间值[0];
       "DB".检测数据.液位实际值 := "DB".检测数据.中间值[1];
   END_IF;
END_REGION
END_FUNCTION

ORGANIZATION_BLOCK "Main"   // OB1, LAD, ProgramCycle
TITLE = "Main Program Sweep (Cycle)"
{ S7_Optimized_Access := 'TRUE' }
VERSION : 0.1
   VAR_INPUT
      Initial_Call : Bool;   // Initial call of this OB
      Remanence : Bool;   // =True, if remanent data are available
   END_VAR
BEGIN

REGION Network 1
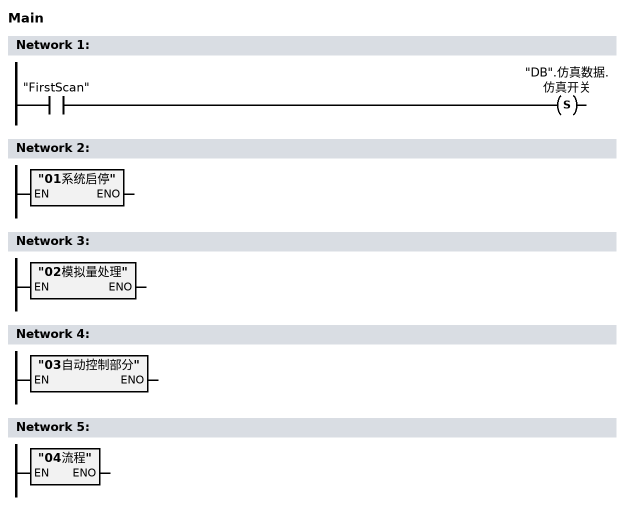
   RUNG wire#powerrail
      Contact( "FirstScan" )
      S_Coil( "DB".仿真数据.仿真开关 )
   END_RUNG
   // the same network as SCL:
   IF "FirstScan" THEN "DB".仿真数据.仿真开关 := TRUE; END_IF;
END_REGION

REGION Network 2
   RUNG wire#powerrail
      "01系统启停"()
   END_RUNG
   // the same network as SCL:
   "01系统启停"();
END_REGION

REGION Network 3
   RUNG wire#powerrail
      "02模拟量处理"()
   END_RUNG
   // the same network as SCL:
   "02模拟量处理"();
END_REGION

REGION Network 4
   RUNG wire#powerrail
      "03自动控制部分"()
   END_RUNG
   // the same network as SCL:
   "03自动控制部分"();
END_REGION

REGION Network 5
   RUNG wire#powerrail
      "04流程"()
   END_RUNG
   // the same network as SCL:
   "04流程"();
END_REGION
END_ORGANIZATION_BLOCK

(* ===== HMI "HMI_RT_1" =====
system functions are stored by id; their names below are inferred from use
connection "HMI_连接_1": ETHERNET, S7_1200_OMS

HMI tags "默认变量表"
   "DB_仿真数据_传送带" : Int = PLC "DB".仿真数据.传送带, 100 ms
   "DB_仿真数据_罐子_X" : Int = PLC "DB".仿真数据.罐子.X, 100 ms
   "DB_仿真数据_罐子_Y" : Int = PLC "DB".仿真数据.罐子.Y, 100 ms
   "DB_仿真数据_灌装1_气缸" : Int = PLC "DB".仿真数据.吹气.气缸, 100 ms
   "DB_仿真数据_灌装2_液位" : Int = PLC "DB".仿真数据.灌装.液位, 100 ms
   "DB_仿真数据_灌装2_气缸" : Int = PLC "DB".仿真数据.灌装.气缸, 100 ms
   "DB_HMI按键_启动" : Bool = PLC "DB".HMI按键.启动, 100 ms
   "DB_HMI按键_停止" : Bool = PLC "DB".HMI按键.停止, 100 ms
   "灌装1气缸上限位" : Bool = PLC 吹气气缸上限位 AT %I1.1, 100 ms
   "灌装1气缸下限位" : Bool = PLC 吹气气缸下限位 AT %I1.2, 100 ms
   "灌装2气缸上限位" : Bool = PLC 灌装气缸上限位 AT %I1.3, 100 ms
   "灌装2气缸下限位" : Bool = PLC 灌装气缸下限位 AT %I1.4, 100 ms
   "DB_检测数据_称重实际值" : Real = PLC "DB".检测数据.称重实际值, 100 ms
   "DB_检测数据_液位仿真值" : Real = PLC "DB".检测数据.液位仿真值, 100 ms
   "DB_仿真数据_拧盖_盖子显示" : Bool = PLC "DB".仿真数据.拧盖.盖子显示, 100 ms
   "DB_仿真数据_拧盖_气缸" : Int = PLC "DB".仿真数据.拧盖.气缸, 100 ms
   "DB_仿真数据_拧盖_拧盖进度" : Int = PLC "DB".仿真数据.拧盖.拧盖进度, 100 ms
   "拧盖气缸上限位" : Bool = PLC 拧盖气缸上限位 AT %I1.5, 100 ms
   "拧盖气缸下限位" : Bool = PLC 拧盖气缸下限位 AT %I2.0, 100 ms
   "到达灌装位置1" : Bool = PLC 到达称重吹气位置 AT %I0.2, 100 ms
   "到达灌装位置2" : Bool = PLC 到达灌装位置 AT %I0.3, 100 ms
   "到达拧盖位置" : Bool = PLC 到达拧盖位置 AT %I0.4, 100 ms
   "到达标签投放位置" : Bool = PLC 到达标签投放位置 AT %I1.0, 100 ms
   "DB_仿真数据_标签投放_小标显示" : Bool = PLC "DB".仿真数据.标签投放.小标显示, 100 ms
   "DB_仿真数据_标签投放_大标显示" : Bool = PLC "DB".仿真数据.标签投放.大标显示, 100 ms
   "DB_仿真数据_标签投放_标签Y" : Int = PLC "DB".仿真数据.标签投放.标签Y, 100 ms
   "DB_仿真数据_热缩_热缩进度" : Int = PLC "DB".仿真数据.热缩.热缩进度, 100 ms
   "DB_仿真数据_清洗_清洗进度" : Int = PLC "DB".仿真数据.清洗.清洗进度, 100 ms
   "DB_仿真数据_消毒_消毒进度" : Int = PLC "DB".仿真数据.消毒.消毒进度, 100 ms
   "到达包装热缩位置" : Bool = PLC 到达包装热缩位置 AT %I0.5, 100 ms
   "到达清洗位置" : Bool = PLC 到达清洗位置 AT %I0.6, 100 ms
   "到达消毒位置" : Bool = PLC 到达消毒位置 AT %I0.7, 100 ms
   "DB_状态_流程" : Int = PLC "DB".状态.流程, 100 ms
   "运行指示灯" : Bool = PLC 运行指示灯 AT %Q0.0, 100 ms
   "DB_HMI按键_复位" : Bool = PLC "DB".HMI按键.复位, 100 ms
   "DB_HMI按键_仿真瓶子质量超重" : Bool = PLC "DB".HMI按键.仿真瓶子质量超重, 100 ms
   "DB_HMI按键_仿真瓶子质量过低" : Bool = PLC "DB".HMI按键.仿真瓶子质量过低, 100 ms
   "瓶子异常示灯" : Bool = PLC 瓶子异常示灯 AT %Q2.2, 100 ms
   "有杂物指示灯" : Bool = PLC 有杂物指示灯 AT %Q2.3, 100 ms

graphic list "传送带": 0 '图形_3'; 1 '图形_4'

screen "画面_1" 800x480
   SymbolLibrary "符号库_6" at 492,50 size 18x84
   SymbolLibrary "符号库_5" at 493,121 size 16x46
   SymbolLibrary "符号库_8" at 679,58 size 24x66
   SymbolLibrary "符号库_2" at 665,120 size 52x30
   Group "Group" at 492,50 size 18x117
      DirectMovement <- "DB_仿真数据_灌装2_气缸"
   Bar "棒图_1" at 145,176 size 31x43; MinimumValue 0; MaximumValue 100
      DirectMovement <- "DB_仿真数据_罐子_X"
      DirectMovement <- "DB_仿真数据_罐子_Y"
      ProcessValue <- "DB_仿真数据_灌装2_液位"
   GraphicIOField "图形 I/O 域_1" at 744,218 size 40x40; PictureList "传送带"
      ProcessValue <- "DB_仿真数据_传送带"
   GraphicIOField "图形 I/O 域_2" at 129,218 size 40x40; PictureList "传送带"
      ProcessValue <- "DB_仿真数据_传送带"
   Ellipse "椭圆_1" at 145,175 size 31x5
      DirectMovement <- "DB_仿真数据_罐子_X"
      DirectMovement <- "DB_仿真数据_罐子_Y"
      Visibility <- "DB_仿真数据_拧盖_盖子显示"
   GraphicIOField "图形 I/O 域_3" at 744,418 size 40x40; PictureList "传送带"
      ProcessValue <- "DB_仿真数据_传送带"
   GraphicIOField "图形 I/O 域_4" at 129,418 size 40x40; PictureList "传送带"
      ProcessValue <- "DB_仿真数据_传送带"
   SymbolLibrary "符号库_3" at 460,50 size 83x71
   Group "Group_1" at 665,58 size 52x92
      DirectMovement <- "DB_仿真数据_拧盖_气缸"
   SymbolLibrary "符号库_9" at 666,50 size 50x67
   Bar "棒图_2" at 653,224 size 76x19; MinimumValue 0; MaximumValue 100
      ProcessValue <- "DB_仿真数据_拧盖_拧盖进度"
   Rectangle "矩形_3" at 335,148 size 17x9
      Appearance <- "灌装1气缸下限位"
   Rectangle "矩形_4" at 335,116 size 17x9
      Appearance <- "灌装1气缸上限位"
   Rectangle "矩形_5" at 526,148 size 17x9
      Appearance <- "灌装2气缸下限位"
   Rectangle "矩形_6" at 526,116 size 17x9
      Appearance <- "灌装2气缸上限位"
   Rectangle "矩形_7" at 725,148 size 17x9
      Appearance <- "拧盖气缸下限位"
   Rectangle "矩形_8" at 725,116 size 17x9
      Appearance <- "拧盖气缸上限位"
   Rectangle "矩形_9" at 302,246 size 17x9
      Appearance <- "到达灌装位置1"
   Rectangle "矩形_10" at 493,246 size 17x9
      Appearance <- "到达灌装位置2"
   Rectangle "矩形_11" at 683,246 size 17x9
      Appearance <- "到达拧盖位置"
   IOField "I/O 域_1" at 273,224 size 76x19; FormatPattern 999
      ProcessValue <- "DB_检测数据_称重实际值"
   IOField "I/O 域_2" at 464,224 size 76x19; FormatPattern 999
      ProcessValue <- "DB_检测数据_液位仿真值"
   TextField "文本域_4" at 334,222 size 14x19; Text 'g'
   TextField "文本域_5" at 526,224 size 14x19; Text '%'
   GraphicView "图形视图_1" at 294,80 size 33x77; Picture "图形_1"
      DirectMovement <- "DB_仿真数据_灌装1_气缸"
   SymbolLibrary "符号库_1" at 269,50 size 83x71
   Rectangle "矩形_12" at 302,446 size 17x9
      Appearance <- "到达标签投放位置"
   SymbolLibrary "符号库_11" at 287,339 size 48x19
   SymbolLibrary "符号库_10" at 286,288 size 50x56
   Rectangle "矩形_13" at 403,446 size 17x9
      Appearance <- "到达包装热缩位置"
   Rectangle "矩形_14" at 553,446 size 17x9
      Appearance <- "到达清洗位置"
   Rectangle "矩形_15" at 683,446 size 17x9
      Appearance <- "到达消毒位置"
   TextField "文本域_1" at 280,26 size 61x17; Text '称重吹气'
   TextField "文本域_2" at 471,26 size 61x17; Text '液体罐装'
   TextField "文本域_3" at 662,26 size 61x17; Text '封装盖盖'
   TextField "文本域_6" at 295,264 size 33x17; Text '标签'
   TextField "文本域_7" at 395,264 size 33x17; Text '热缩'
   TextField "文本域_8" at 545,264 size 33x17; Text '清洗'
   TextField "文本域_9" at 675,264 size 33x17; Text '消毒'
   GraphicView "图形视图_2" at 145,116 size 31x20; Picture "图形_5"
      DirectMovement <- "DB_仿真数据_罐子_X"
      Visibility <- "DB_仿真数据_标签投放_小标显示"
      DirectMovement <- "DB_仿真数据_标签投放_标签Y"
   GraphicView "图形视图_3" at 142,116 size 37x20; Picture "图形_5"
      DirectMovement <- "DB_仿真数据_罐子_X"
      Visibility <- "DB_仿真数据_标签投放_大标显示"
      DirectMovement <- "DB_仿真数据_标签投放_标签Y"
   Bar "棒图_3" at 389,372 size 44x47; MinimumValue 0; MaximumValue 100
      ProcessValue <- "DB_仿真数据_热缩_热缩进度"
   Bar "棒图_4" at 539,372 size 44x47; MinimumValue 0; MaximumValue 100
      ProcessValue <- "DB_仿真数据_清洗_清洗进度"
   Bar "棒图_5" at 669,372 size 44x47; MinimumValue 0; MaximumValue 100
      ProcessValue <- "DB_仿真数据_消毒_消毒进度"
   Button "按钮_1" at 22,27 size 74x27; TextOff '启动'
      on Press: function_b14e0dd5("DB_HMI按键_启动", 0)
      Appearance <- "运行指示灯"
   Button "按钮_2" at 22,66 size 74x27; TextOff '停止'
      on Press: function_b14e0dd5("DB_HMI按键_停止", 0)
      Appearance <- "运行指示灯"
   Button "按钮_10" at 22,105 size 74x27; TextOff '复位'
      on Press: function_b14e0dd5("DB_HMI按键_复位", 0)
   Button "按钮_3" at 22,173 size 74x27; TextOff '称重吹气'
      Appearance <- "DB_状态_流程"
   Button "按钮_4" at 22,214 size 74x27; TextOff '液体罐装'
      Appearance <- "DB_状态_流程"
   Button "按钮_5" at 22,256 size 74x27; TextOff '封装盖盖'
      Appearance <- "DB_状态_流程"
   Button "按钮_6" at 22,298 size 74x27; TextOff '标签'
      Appearance <- "DB_状态_流程"
   Button "按钮_7" at 22,340 size 74x27; TextOff '热缩'
      Appearance <- "DB_状态_流程"
   Button "按钮_8" at 22,382 size 74x27; TextOff '清洗'
      Appearance <- "DB_状态_流程"
   Button "按钮_9" at 22,424 size 74x27; TextOff '消毒'
      Appearance <- "DB_状态_流程"
   Button "按钮_11" at 142,27 size 106x27; TextOff '超重仿真'
      on Click: InvertBit("DB_HMI按键_仿真瓶子质量超重")
      Appearance <- "DB_HMI按键_仿真瓶子质量超重"
   Button "按钮_12" at 142,66 size 106x27; TextOff '过轻仿真'
      on Click: InvertBit("DB_HMI按键_仿真瓶子质量过低")
      Appearance <- "DB_HMI按键_仿真瓶子质量过低"
   Button "按钮_13" at 271,55 size 79x33; TextOff '瓶子异常'
      Visibility <- "瓶子异常示灯"
   Button "按钮_14" at 271,55 size 79x33; TextOff '有杂物'
      Visibility <- "有杂物指示灯"
*)